ABB RobotStudio station: Current1_20190820-162655.rsstn

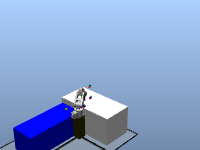
Station Solution2 (saved by RobotStudio 7.0.8504.151)
Controller IRB_120_3kg_0.58m, task T_ROB1: task frame (RAPID world) sits at (0, 0, 580.99) mm in the station
Controller IRB_120_3kg_0.58m
  mechanical unit ROB_1: IRB120_3_58__01, 6 joints, base frame (0, 0, 0) mm
Layout (positions relative to the parent item):
  - IRB120_3_58__01 [mechanism, from Robots\IRB120_3_58_G_01.rslib] at (0, 0, 580.99) mm; joint values [0.4812, 0.7783, -0.0517, 0, 0.8442, -0.1045] (rad or m)
  - ABBconvayor [part]
  - ABBstand [part]
  - ABBtable [part]
Collision set CollisionSet_1: IRB120_3_58__01 against ABBtable, ABBconvayor, near miss 0 m
Targets, tools, work objects and paths stored in the station, written as RAPID:
! task T_ROB1
MODULE MattServer
  PROC main()
    MainServer;
  ENDPROC
  PROC MainServer()
    ListenForAndAcceptConnection;
    WaitForMessage;
    CloseConnection;
  ENDPROC
  PROC WaitForMessage()
    MattMain;
  ENDPROC
  PROC ListenForAndAcceptConnection()
  ENDPROC
  PROC CloseConnection()
  ENDPROC
ENDMODULE

! task T_ROB1
MODULE Vacuum
  CONST robtarget pConvHome:=[[0,409,22],[0,-0.7071068,0.7071068,0],[0,0,0,0],[9E+09,9E+09,9E+09,9E+09,9E+09,9E+09]];
  PROC testMove()
    MoveL pConvHome,v100,fine,tSCup;
  ENDPROC
  PROC turnOnVacuum()
    Set DO10_1;
  ENDPROC
  PROC turnOffVacuum()
    turnOffGripper;
    Reset DO10_1;
  ENDPROC
  PROC turnOnGripper()
  ENDPROC
  PROC turnOffGripper()
    Reset DO10_2;
  ENDPROC
  PROC Vacmain()
    turnOnVacuum;
    WaitTime 5;
    turnOnGripper;
    WaitTime 2;
    turnOffGripper;
    WaitTime 2;
    turnOffVacuum;
    testMove;
  ENDPROC
ENDMODULE

! task T_ROB1
MODULE MattMove
  PROC PrintCurPose()
  ENDPROC
  PROC PrintCurJoint()
  ENDPROC
  PROC MoveJMatt()
    MoveJ pDemand,v100,fine,tSCup;
    MoveJ pTableHome,v100,fine,tSCup;
  ENDPROC
  PROC MattMain()
    MoveToCalibPos;
    PrintCurPose;
    MattTurnVacOff;
    WaitTime 2.0;
    MoveToCalibPos;
  ENDPROC
  PROC MattTurnVacOn()
    SetDO DO10_1,1;
    SetDO DO10_2,1;
  ENDPROC
  PROC MattTurnVacOff()
    SetDO DO10_2,0;
    SetDO DO10_1,0;
  ENDPROC
ENDMODULE

! task T_ROB1
MODULE MTRN_Rob_Data
  PERS wobjdata wTable:=[FALSE,TRUE,"",[[175,0,147],[1,0,0,0]],[[0,0,0],[1,0,0,0]]];
  PERS wobjdata wConv:=[FALSE,TRUE,"",[[50,184,22],[0.5,-0.5,0.5,0.5]],[[1,1,1],[1,0,0,0]]];
  CONST robtarget pTableHome:=[[175,0,147],[0,0,-1,0],[0,0,0,0],[9E+09,9E+09,9E+09,9E+09,9E+09,9E+09]];
  CONST jointtarget jtCalibPos:=[[0,0,0,0,0,0],[9E+09,9E+09,9E+09,9E+09,9E+09,9E+09]];
  CONST jointtarget jtHomePos:=[[-90,0,0,0,0,0],[9E+09,9E+09,9E+09,9E+09,9E+09,9E+09]];
  PERS tooldata tSCup:=[TRUE,[[0,0,65],[1,0,0,0]],[0.5,[0,0,20],[1,0,0,0],0,0,0]];
ENDMODULE

! task T_ROB1
MODULE MTRN_Rob_Proc
  PROC MoveToCalibPos()
    MoveAbsJ jtCalibPos,v400,fine,tool0;
  ENDPROC
  PROC MoveToHomePos()
    MoveAbsJ jtHomePos,v400,fine,tool0;
  ENDPROC
ENDMODULE

! task T_ROB1
MODULE MTRN4230_IO_Sample
  PROC TurnVacOn()
    SetDO DO10_1,1;
  ENDPROC
  PROC TurnVacOff()
    SetDO DO10_1,0;
  ENDPROC
  PROC TurnConOnSafely()
  ENDPROC
  PROC TurnConOff()
    SetDO DO10_3,0;
  ENDPROC
  PROC MainIO()
    TurnVacOn;
    WaitTime 2;
    TurnVacOff;
    TurnConOnSafely;
    WaitTime 2;
    TurnConOff;
  ENDPROC
ENDMODULE

